FUNCTION_BLOCK EL4008
VAR
	_io : EL4xx8_Data;
	{attribute addProperty Name "WcState"}
	_wcState : WcStateBase;
	{attribute addProperty Name "Info data"}
	_infoData : InfoDataAds;
END_VAR

PROPERTY IO : REFERENCE TO EL4xx8_Data
GET
IO REF= _io;
END_GET
END_PROPERTY

PROPERTY WcState : REFERENCE TO WcStateBase
GET
WcState REF= _wcState;
END_GET
END_PROPERTY

END_FUNCTION_BLOCK

(* stored: Version 1.1.0.1, ProductVersion 3.1.4024.9
   POU EL4008: Id {93ea128e-a8f1-05c3-1afa-1f71d95fd50c}, SpecialFunc None
   Property IO: Id {b2505f9d-9374-0141-19cc-4058fe973104}
   Get Get: Id {aca742a9-d132-0160-02e5-a834a2444ac6}
   Property WcState: Id {aadfe4a1-5139-02c6-3d73-a56a6b770a54}
   Get Get: Id {d905d488-6e50-023b-0c5c-f7ffa6b9cdca} *)
